(* CoDeSys 2.3.9.35 project: SANALOGICA1.pro *)
(* Author: Altus *)
(* Libraries: DU35x.lib 7.7.11 15:59:13, Navigation.lib 15.7.11 10:06:00, SysLibTargetVisu.lib 26.11.08 09:53:28, Standard.lib 26.11.08 09:46:20, Iecsfc.lib 26.11.08 09:46:14, SYSLIBCALLBACK.LIB 26.11.08 09:53:30 *)

(* PLC configuration (modules and I/O channels)
Comunicação [Comunica] node 0, in %IB0 out %QB0
  COM1 [COM1] node 0, in %IB0 out %QB0 {BaudRate = 115200; Paridade = Sem Paridade; StopBits = 1 Stop Bit; Modem = Sem RTS/CTS; Delay = 5}
    MToolIEC [Codesys] node 0, in %IB0 out %QB0
  COM2 [COM2] node 1, in %IB0 out %QB0 {BaudRate = 115200; Paridade = Sem Paridade; StopBits = 1 Stop Bit; Modem = Sem RTS/CTS; Delay = 5}
    Desabilitada [Desabilitado485] node 0, in %IB0 out %QB0
Entradas Digitais 0 [Entradas0] node 0, in %IW0 out %QB0
  I00 AT %IX0.0 [BitInput] I0.0
  I01 AT %IX0.1 [BitInput] I0.1
  I02 AT %IX0.2 [BitInput] I0.2
  I03 AT %IX0.3 [BitInput] I0.3
  I04 AT %IX0.4 [BitInput] I0.4
  I05 AT %IX0.5 [BitInput] I0.5
  I06 AT %IX0.6 [BitInput] I0.6
  I07 AT %IX0.7 [BitInput] I0.7
  I08 AT %IX0.8 [BitInput] I0.8
Entradas Digitais 1 [Entradas1] node 0, in %IW1 out %QB0
  I10 AT %IX1.0 [BitInput] I1.0
  I11 AT %IX1.1 [BitInput] I1.1
  I12 AT %IX1.2 [BitInput] I1.2
  I13 AT %IX1.3 [BitInput] I1.3
  I14 AT %IX1.4 [BitInput] I1.4
  I15 AT %IX1.5 [BitInput] I1.5
  I16 AT %IX1.6 [BitInput] I1.6
  I17 AT %IX1.7 [BitInput] I1.7
  I18 AT %IX1.8 [BitInput] I1.8
Entradas Digitais 2 [Entradas2] node 0, in %IW2 out %QB0
  I20 AT %IX2.0 [BitInput] I2.0
  I21 AT %IX2.1 [BitInput] I2.1
AI0 AT %IW4 [WordInput] AI0 {TipoAnalogica = Tensão 0-10V; FiltroAnalogica = Filtro 0 - AI=2ms  / AV=90ms; FundoEscala = 10}
AI1 AT %IW5 [WordInput] AI1 {TipoAnalogica = Channel Disable; FiltroAnalogica = Filter 0 - AI=2ms  / AV=90ms; FundoEscala = 0}
AI2 AT %IW6 [WordInput] AI2 {TipoAnalogica = Channel Disable; FiltroAnalogica = Filter 0 - AI=2ms  / AV=90ms; FundoEscala = 0}
AI3 AT %IW7 [WordInput] AI3 {TipoAnalogica = Channel Disable; FiltroAnalogica = Filter 0 - AI=2ms  / AV=90ms; FundoEscala = 0}
Bloco 0 [Bloco0] node 0, in %IB16 out %QB0
  Desabilitado [DesabilitadoBloco0] node 0, in %IB16 out %QB0
Bidirecional [BidirecionalBloco1] node 0, in %IB16 out %QB0 {ContagemBidirecional = Quadratura 2x}
Contador 0 [EntradaConfContador0] node 0, in %IB16 out %QB0 {EntradaConfiguravelContador = Desabilitada}
Contador 2 [EntradaConfContador2] node 0, in %IB16 out %QB0 {EntradaConfiguravelContador = Zeramento}
Saídas Digitais 0 [Saidas0] node 0, in %IW0 out %QW0
  Q00 AT %QX0.0 [BitOutput] Q0.0
  Q01 AT %QX0.1 [BitOutput] Q0.1
  Q02 AT %QX0.2 [BitOutput] Q0.2
  Q03 AT %QX0.3 [BitOutput] Q0.3
  Q04 AT %QX0.4 [BitOutput] Q0.4
  Q05 AT %QX0.5 [BitOutput] Q0.5
  Q06 AT %QX0.6 [BitOutput] Q0.6
  Q07 AT %QX0.7 [BitOutput] Q0.7
Saídas Digitais 1 [Saidas1] node 0, in %IW0 out %QW1
  Q10 AT %QX1.0 [BitOutput] Q1.0
  Q11 AT %QX1.1 [BitOutput] Q1.1
  Q12 AT %QX1.2 [BitOutput] Q1.2
  Q13 AT %QX1.3 [BitOutput] Q1.3
  Q14 AT %QX1.4 [BitOutput] Q1.4
  Q15 AT %QX1.5 [BitOutput] Q1.5
  Q16 AT %QX1.6 [BitOutput] Q1.6
  Q17 AT %QX1.7 [BitOutput] Q1.7
AO0 AT %QW3 [WordOutput] AO0 {TipoAnalogica = Channel Disable; FundoEscala = 0}
AO1 AT %QW4 [WordOutput] AO1 {TipoAnalogica = Tensão 0-10V; FundoEscala = 10}
Saída Rápida 0 Desabilitada [DesabilitadoF0] node 0, in %IB0 out %QB10
PTO [PTOF1] node 1, in %IB0 out %QB10 {RampaPTO = Trapezoidal}
Saídas Comum de Contador [SaidasContador] node 2, in %IB0 out %QB10
  Saída do Bloco 0 Desabilitada [DesabilitadoSaidaBloco0] node 0, in %IB0 out %QB10
  Saída do Bloco 1 Desabilitada [DesabilitadoSaidaBloco1] node 1, in %IB0 out %QB10
Eventos Externos [Eventos] node 2, in %IB13 out %QB6
  Evento Temporizado [TimerEvent] node 0, in %IB13 out %QB6 {Intervalo = 10}
*)

(* Task configuration *)
TASK PRINCIPAL (PRIORITY := 1, INTERVAL := T#1ms);
	PLC_PRG();
END_TASK
TASK NAVIGATION (PRIORITY := 1, INTERVAL := T#20ms);
	NAVEGA();
END_TASK
TASK VISUALIZATION (PRIORITY := 1, INTERVAL := T#500ms);
	MAINTARGETVISU_PAINT_CODE
END_TASK
TASK KEYBOARD_USAGE (PRIORITY := 1, INTERVAL := T#20ms);
	MAINTARGETVISU_INPUT_CODE
END_TASK

(* POU PLC_PRG, LD *)
PROGRAM PLC_PRG
VAR
	FREQ AT %MD1652: DWORD;		(*FREQUENCIA DO SINA DE SAIDA*)
	PLS_TOT AT %MD1653: DWORD;	(*NUMERO DE PULSOS TOTAL*)
	PLS_RAMP AT %MD1654: DWORD; (*NUMERO DE PULSOS POR RAMPA DE ACELARACAO/DESACELERACAO*)
	SENT_ROTA AT %QX0.2: BOOL := 0;			(*SENTIDO DE ROTAÇÃO DO MOTOR 0= HORARIO 1= ANT-HORARIO*)
	HAB_MOTOR AT %QX0.3: BOOL := 0;			(*HABILITA O MOTOR 1=BONINAS PERMANECE ENERGIZADAS 0=BONINAS ENERGIZADAS PENAS DURANTE O MOVIMENTO*)
	PLS_QTD AT %QX0.4: BOOL := 0;			(*QUANTIDADE DE PULSOS 0= 200 PULOS PARA UMA VOLTA 1=400 PULOS PARA UMA VOLTA*)

	START_MOTOR AT %MX3314.2: BOOL := 0; (*ACIONA O DISPARO DOS PULSOS NA SAIDA RAPAIDA*)
	STOP_MOTOR AT %MX3314.3: BOOL := 0; (*PARA O DISPARO DOS PULSOS NA SAIDA RAPAIDA*)

	CONTADOR AT %MD1633:DWORD;(*ENTRADA RAPIDA PARA ACESSAR A O CONTADOR 1 LIGADO AO ENCODER*)
	ZERA AT %QX0.0: BOOL;(*SAIDA UTILIZADO PARA ZERAR O CONTADOR*)
	HABILITA AT %IX0.0: BOOL := 0;
	HABILITA2 AT %IX0.1: BOOL := 0;
	POT AT %IW4: WORD := 0;(*ENTRADA DA LETURA DO POTENCIOMENTRO*)
	DISPLAY: REAL:=0;
	PLS_CONT: REAL; (*NUMERO DE PULSOS CONTADOS*)
	AUX_PLS_CONT: DWORD;
	ROTACAO: REAL:=0;
	RPM: REAL:=0;
	SAIDA AT %QW4: WORD := 0;
	MN AT %IX0.2: BOOL;
	MR AT %IX0.3: BOOL;
	MT AT %IX0.4: BOOL;
	AUX_TEMP_PLS_READ: BOOL;
	AUX2: BOOL;
	AUX3: BOOL;
	AUX4: BOOL;
	TEMP_ROT_HORARIO: TON;
	TEMP_ROT_ANT_HORARIO: TOF;
	AUXPOT: DWORD;
	SMN: BOOL;
	SMR: BOOL;
	SMT: BOOL;
	TEMP_PLS_READ: TON;
	LIGA: AT %IX0.0: BOOL :=0;
	LIGADO: BOOL;
	DESLIGA: AT %IX0.1: BOOL := 0;
	AUX_RPM: BOOL;
	PARA: BOOL;
END_VAR
VAR (* helpers for the ST form of the networks *)
	_p1 : BOOL;
	_p2 : BOOL;
END_VAR
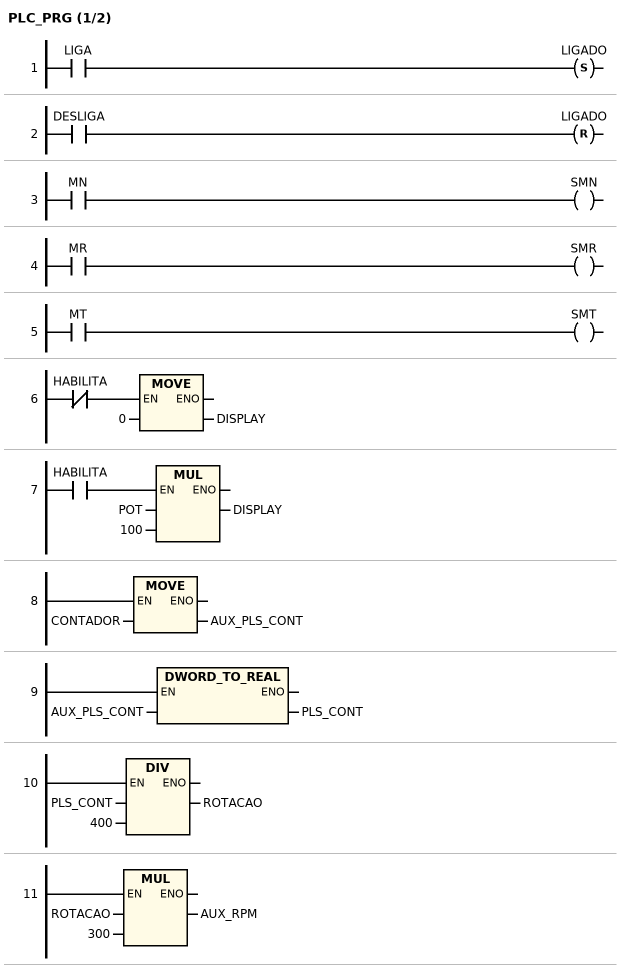
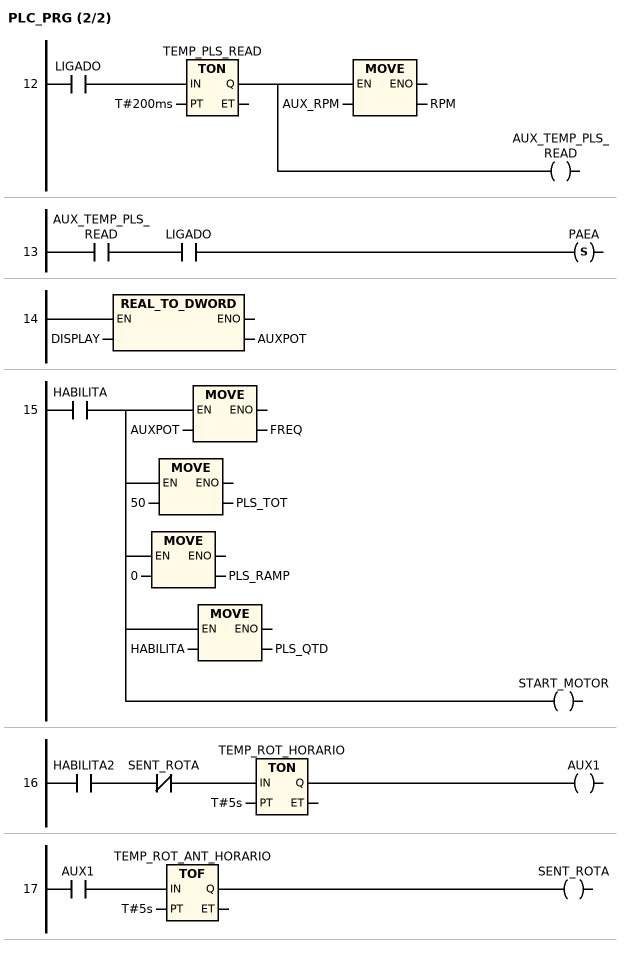
_LD_ (* Ladder Diagram *)
NETWORK 1
	[LIGA] --- (S LIGADO)
NETWORK 2
	[DESLIGA] --- (R LIGADO)
NETWORK 3
	[MN] --- (SMN)
NETWORK 4
	[MR] --- (SMR)
NETWORK 5
	[MT] --- (SMT)
NETWORK 6
	[/HABILITA]
		EN --- MOVE(0) => DISPLAY
NETWORK 7
	[HABILITA]
		EN --- MUL(POT, 100) => DISPLAY
NETWORK 8
	*
		EN --- MOVE(CONTADOR) => AUX_PLS_CONT
NETWORK 9
	*
		EN --- DWORD_TO_REAL(AUX_PLS_CONT) => PLS_CONT
NETWORK 10
	*
		EN --- DIV(PLS_CONT, 400) => ROTACAO
NETWORK 11
	*
		EN --- MUL(ROTACAO, 300) => AUX_RPM
NETWORK 12
	[LIGADO] - TEMP_PLS_READ:TON(IN: *, PT: T#200ms) --- (AUX_TEMP_PLS_READ)
		EN --- MOVE(AUX_RPM) => RPM
NETWORK 13
	[AUX_TEMP_PLS_READ] - [LIGADO] --- (S PAEA)
NETWORK 14
	*
		EN --- REAL_TO_DWORD(DISPLAY) => AUXPOT
NETWORK 15
	[HABILITA] --- (START_MOTOR)
		EN --- MOVE(AUXPOT) => FREQ
		EN --- MOVE(50) => PLS_TOT
		EN --- MOVE(0) => PLS_RAMP
		EN --- MOVE(HABILITA) => PLS_QTD
NETWORK 16
	[HABILITA2] - [/SENT_ROTA] - TEMP_ROT_HORARIO:TON(IN: *, PT: T#5s) --- (AUX1)
NETWORK 17
	[AUX1] - TEMP_ROT_ANT_HORARIO:TOF(IN: *, PT: T#5s) --- (SENT_ROTA)
_END_LD_
(* the same logic as Structured Text *)
(* Network 1 *)
IF LIGA THEN LIGADO := TRUE; END_IF;
(* Network 2 *)
IF DESLIGA THEN LIGADO := FALSE; END_IF;
(* Network 3 *)
SMN := MN;
(* Network 4 *)
SMR := MR;
(* Network 5 *)
SMT := MT;
(* Network 6 *)
IF NOT HABILITA THEN
	DISPLAY := 0;
END_IF;
(* Network 7 *)
IF HABILITA THEN
	DISPLAY := POT * 100;
END_IF;
(* Network 8 *)
AUX_PLS_CONT := CONTADOR;
(* Network 9 *)
PLS_CONT := DWORD_TO_REAL(AUX_PLS_CONT);
(* Network 10 *)
ROTACAO := PLS_CONT / 400;
(* Network 11 *)
AUX_RPM := ROTACAO * 300;
(* Network 12 *)
TEMP_PLS_READ(IN := LIGADO, PT := T#200ms);
_p1 := TEMP_PLS_READ.Q;
IF _p1 THEN
	RPM := AUX_RPM;
END_IF;
AUX_TEMP_PLS_READ := _p1;
(* Network 13 *)
IF AUX_TEMP_PLS_READ AND LIGADO THEN PAEA := TRUE; END_IF;
(* Network 14 *)
AUXPOT := REAL_TO_DWORD(DISPLAY);
(* Network 15 *)
_p2 := HABILITA;
IF _p2 THEN
	FREQ := AUXPOT;
	PLS_TOT := 50;
	PLS_RAMP := 0;
	PLS_QTD := HABILITA;
END_IF;
START_MOTOR := _p2;
(* Network 16 *)
TEMP_ROT_HORARIO(IN := HABILITA2 AND NOT SENT_ROTA, PT := T#5s);
AUX1 := TEMP_ROT_HORARIO.Q;
(* Network 17 *)
TEMP_ROT_ANT_HORARIO(IN := AUX1, PT := T#5s);
SENT_ROTA := TEMP_ROT_ANT_HORARIO.Q;
END_PROGRAM

(* POU NAVEGA, ST *)
PROGRAM NAVEGA
VAR
	ControleTelas : NAVIGATION;
	ListaTelas 	: ARRAY [0..30] OF STRING(10);
END_VAR
(* Adiciona a tela MAIN como tela principal *)
ListaTelas[0] := 'MAIN';

(* Ativa o controle automático de navegação somente pelo teclado *)
ControleTelas(ENABLE_UPDW := FALSE, VISU_LIST := ListaTelas, UP := FALSE , DOWN := FALSE);
END_PROGRAM

(* Visualisation MAIN
rectangle at (11,7)-(37,17): text "%0.f"; shows PLC_PRG.DISPLAY
*)
